// Mitsubishi GX Works2 project: 실린더응용5   PLC: Q02/Q02H

PROGRAM MAIN
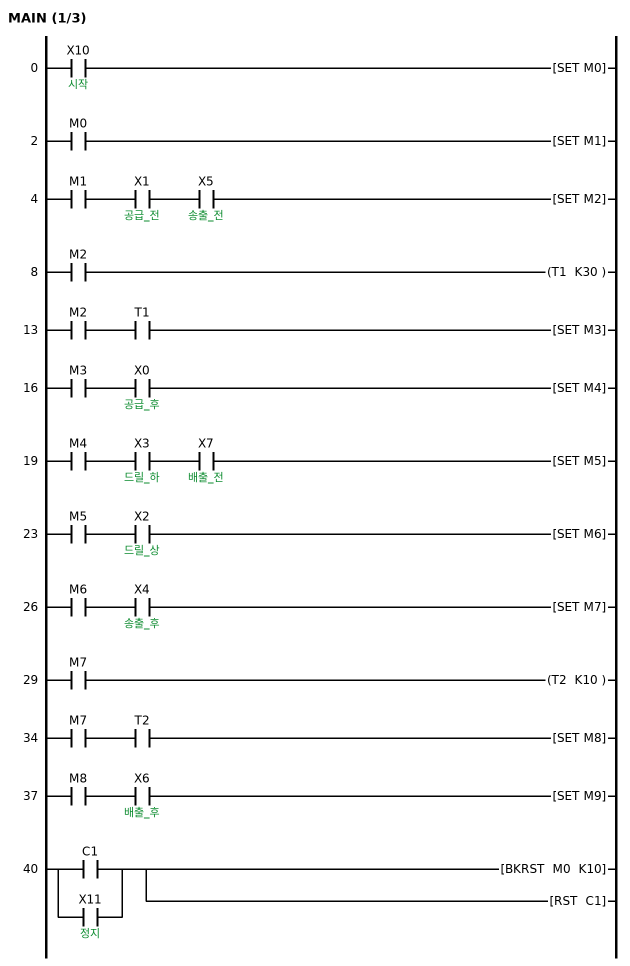
0     LD      X10  ; 시작
      SET     M0
2     LD      M0
      SET     M1
4     LD      M1
      AND     X1  ; 공급_전
      AND     X5  ; 송출_전
      SET     M2
8     LD      M2
      OUT     T1 K30
13    LD      M2
      AND     T1
      SET     M3
16    LD      M3
      AND     X0  ; 공급_후
      SET     M4
19    LD      M4
      AND     X3  ; 드릴_하
      AND     X7  ; 배출_전
      SET     M5
23    LD      M5
      AND     X2  ; 드릴_상
      SET     M6
26    LD      M6
      AND     X4  ; 송출_후
      SET     M7
29    LD      M7
      OUT     T2 K10
34    LD      M7
      AND     T2
      SET     M8
37    LD      M8
      AND     X6  ; 배출_후
      SET     M9
40    LD      C1
      OR      X11  ; 정지
      BKRST   M0 K10
      RST     C1
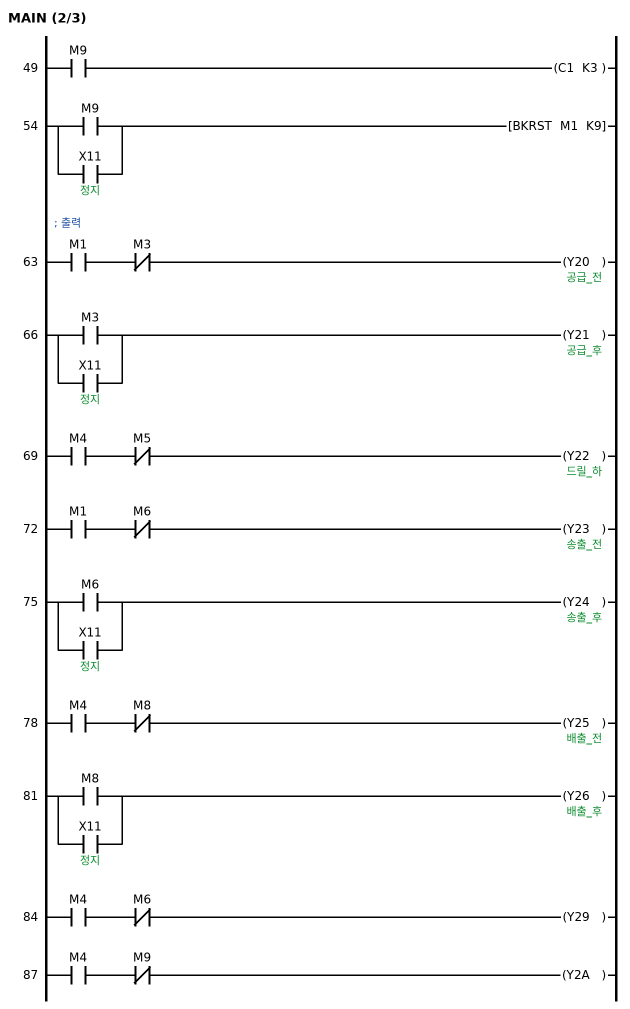
49    LD      M9
      OUT     C1 K3
54    LD      M9
      OR      X11  ; 정지
      BKRST   M1 K9
; 출력
63    LD      M1
      ANI     M3
      OUT     Y20  ; 공급_전
66    LD      M3
      OR      X11  ; 정지
      OUT     Y21  ; 공급_후
69    LD      M4
      ANI     M5
      OUT     Y22  ; 드릴_하
72    LD      M1
      ANI     M6
      OUT     Y23  ; 송출_전
75    LD      M6
      OR      X11  ; 정지
      OUT     Y24  ; 송출_후
78    LD      M4
      ANI     M8
      OUT     Y25  ; 배출_전
81    LD      M8
      OR      X11  ; 정지
      OUT     Y26  ; 배출_후
84    LD      M4
      ANI     M6
      OUT     Y29
87    LD      M4
      ANI     M9
      OUT     Y2A
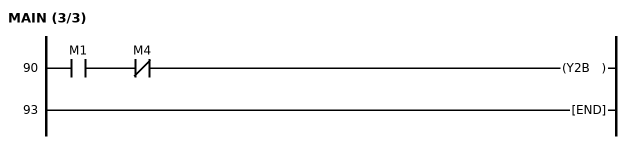
90    LD      M1
      ANI     M4
      OUT     Y2B
93    END
END_PROGRAM
